{attribute 'qualified_only'}
{attribute 'strict'}
{attribute 'to_string'}
TYPE E_AdjustmentStep :
(
    Idle                    := 0,

    MoveXYToWork            := 80,
    LowerZToWork            := 90,
    OpenGripper             := 95,
    PrepareMeasurement      := 100,
    RequestMeasure          := 105,
    WaitMeasureResult       := 110,
    WaitMeasureRetryDelay   := 112,
    EvaluateAdjustment      := 115,
    StartCorrectionXY       := 120,
    WaitCorrectionXY        := 125,
    RequestSecondTighten    := 130,
    WaitSecondTighten       := 135,
    RequestFinalMeasure     := 140,
    WaitFinalMeasure        := 145,
    WaitFinalMeasureRetryDelay := 147,
    EvaluateFinalResult     := 150,
    RequestReworkLoosen     := 155,
    WaitReworkLoosen        := 160,
    CloseGripper            := 170,
    LiftZToSafe             := 180,
    ReturnXYToStandby       := 190,
    WaitDoneAck             := 200,

    Error                   := 900
);
END_TYPE

(* stored: Version 1.1.0.1, ProductVersion 3.1.4026.20
   DUT E_AdjustmentStep: Id {d2db074d-e9dc-4ba1-bcd8-d449f6baf137} *)
